// SIMATIC STEP 7 (V5.x) project test
// CPU: CPU 312
// station: Hardware
// station: SIMATIC 300(1)
// station: P_ADR_BUS
// program: S7 Program(1)

SYMBOL_TABLE
"input 1"	I 0.0	BOOL
"stop"	I 0.1	BOOL
"output 1"	Q 0.0	BOOL
END_SYMBOL_TABLE
